Staubli VAL3: SUB.pjx

Parameters version=s7.2.1 stackSize=5000 millimeterUnit=true
Data file=SUB.dtx
Type name=progItem path=Disk://kernel/template/progItem/progItem.pjx
